TYPE "LubrMotor_Par"
VERSION : 0.1
// Block: LubrMotor_Par
   STRUCT
      EnableCheckRotation : Bool;
      LowLevelCheckTime : Time;
      RotationFbkCheckTime : Time;
   END_STRUCT;

END_TYPE
